{attribute 'pack_mode' := '1'}
TYPE TManBarrelAxisPosition :
STRUCT
		TMove1Step				: TManButton;
		TMoveSectionA			: TManButton;
		TMoveSectionB			: TManButton;
		TMoveSectionC			: TManButton;
		TMoveSectionD			: TManButton;
END_STRUCT
END_TYPE

(* stored: Version 1.1.0.1, ProductVersion 3.1.4022.12
   DUT TManBarrelAxisPosition: Id {95e67fc0-e213-4d86-817b-8d7991dc21b4} *)
